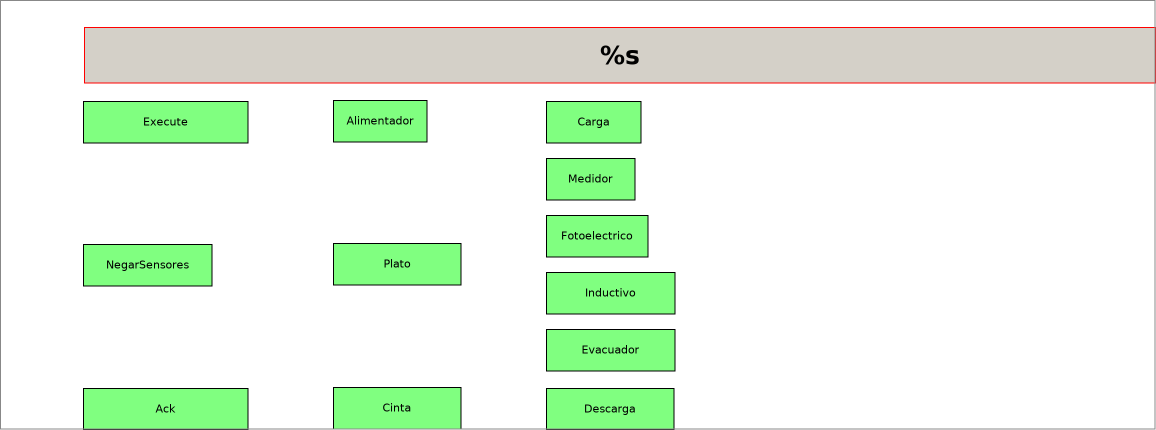
VISUALIZATION FMS205Testing  // 1156x430
VAR_IN_OUT
	
END_VAR
(*VAR
	TestAlimentador
END_VAR^*)
    Rectangle (84,27 1072x56), "%s", text variable: sel(MAIN.fbFMS205.fbPanel.Probando,'Panel de pruebas inactivo','Panel de pruebas ACTIVO')
        toggle MAIN.fbFMS205.fbPanel.Probando
    Rectangle (83,101 165x42), "Execute"
        toggle MAIN.fbFMS205.td.Execute
    Rectangle (83,388 165x42), "Ack"
        tap MAIN.fbFMS205.td.Ack
    Rectangle (333,100 94x42), "Alimentador"
        toggle MAIN.fbFMS205.td.Alime
    Rectangle (546,101 95x42), "Carga"
        toggle MAIN.fbFMS205.td.Carga
    Rectangle (546,158 89x42), "Medidor"
        toggle MAIN.fbFMS205.td.Medid
    Rectangle (546,215 102x42), "Fotoelectrico"
        toggle MAIN.fbFMS205.td.Fotoe
    Rectangle (546,272 129x42), "Inductivo"
        toggle MAIN.fbFMS205.td.Induc
    Rectangle (546,329 129x42), "Evacuador"
        toggle MAIN.fbFMS205.td.Evacu
    Rectangle (546,388 128x42), "Descarga"
        toggle MAIN.fbFMS205.td.Desca
    Rectangle (333,243 128x42), "Plato"
        toggle MAIN.fbFMS205.td.Plato
    Rectangle (83,244 129x42), "NegarSensores"
        tap MAIN.fbFMS205.td.Negar
    Rectangle (333,387 128x42), "Cinta"
        toggle MAIN.fbFMS205.td.Cinta
END_VISUALIZATION

(* stored: Version 1.1.0.1, ProductVersion 3.1.4024.11
   Visu FMS205Testing: Id {d10fef3f-e567-4db8-8634-f52f25296e47} *)
